FUNCTION_BLOCK FB_SolidSamplingModule
VAR_INPUT
END_VAR
VAR_OUTPUT
END_VAR
VAR
END_VAR

END_FUNCTION_BLOCK

(* stored: Version 1.1.0.1
   POU FB_SolidSamplingModule: Id {83628d4f-36fd-490f-a977-5cf01525dad5}, SpecialFunc None *)
